(* IEC 61131-3 sources: Automation-Projects-Portfolio/Project1-TankLevelControl, 7 files *)

(* ---- DUT_Alarms.st ---- *)
TYPE DUT_Alarms :
STRUCT
		// Alarms setpoint
	rSetPointAlarm_HH : REAL := 90.0;
	rSetPointAlarm_H : REAL := 80.0;
	rSetPointAlarm_L : REAL := 20.0;
	rSetPointAlarm_LL : REAL := 10.0;

	//Alarm Status
	xAlarm_HH : BOOL;
	xAlarm_H : BOOL;
	xAlarm_L : BOOL ;
	xAlarm_LL : BOOL;

	//Sensor Fault
	xSensorFault : BOOL;
END_STRUCT
END_TYPE

(* ---- GVLInputs.st ---- *)
VAR_GLOBAL
	rLevelRaw : REAL; //Measured level from level transmitter
	xInletPumpRunFB : BOOL; //Feedback if inlet pump works
	xOutletPumpRunFB : BOOL; //Feedback if outlet pump works
	xEmergencyStop : BOOL := TRUE; //Emergency Button
END_VAR

(* ---- GVLOutputs.st ---- *)
VAR_GLOBAL
	xInletPumpStart : BOOL; //It is inlet pump start signal, if its contactor gets 24V DC from PLC, it will run
	xOutletPumpStart : BOOL; //It is outlet pump start signal, if its contactor gets 24V DC from PLC, it will run
	rValvePosition : REAL; //It is valve position which is decided by PID or an operator
END_VAR

(* ---- FB_ControlValve.st ---- *)
FUNCTION_BLOCK FB_ControlValve
VAR_INPUT
	xAutoMode : BOOL; // Auto = true, manual = false
	rAutoValvePosition : REAL; //Auto Valve position by PID
	rManualValvePosition : REAL; // Manual Valve Position by PID
	xSafetyClose : BOOL; //IF it is true, force valve to stop
END_VAR
VAR_OUTPUT
	rValvePosition : REAL; //ValvePosition is sent to control Valve
END_VAR
VAR
END_VAR

IF xSafetyClose THEN
	rValvePosition := 0.0; // Closed Valve
ELSIF xAutoMode THEN
	rValvePosition := rAutoValvePosition;
ELSE
	rValvePosition := rManualValvePosition;
END_IF

//Limit Valve Position
IF rValvePosition > 100.0 THEN
	rValvePosition := 100.0;
ELSIF rValvePosition < 0.0 THEN
	rValvePosition := 0.0;
END_IF

(* ---- FB_LevelControl.st ---- *)
FUNCTION_BLOCK FB_LevelControl
VAR_INPUT
	xAutoMode : BOOL; // TRUE = Auto FALSE = MANUAL
	rLevel : REAL; //Input from GVLInputs
	rSetPoint : REAL; //Target Level
	rKp : REAL := 2.0; // Proportianl gain in seconds;
	rTn : REAL := 10.0; //Integral time in seconds;
	rTv : REAL := 0.0;// DerivativeTime in seconds
	xResetAlarms : BOOL; //Reset after error is removed
END_VAR
VAR_OUTPUT
	rPidOutput : REAL;
	stAlarms : DUT_Alarms;
END_VAR
VAR
	PID : UTIL.PID;
	fbResetTrigger : R_TRIG; //Function block for reset
	xResetPulse : BOOL;
END_VAR

// 1. Reset for one cycle
fbResetTrigger ( CLK := xResetAlarms, Q => xResetPulse);

// 2. Sensor Fault Detection & Latched Reset
IF (rLevel < -2.0) OR (rLevel > 102.0) THEN
    stAlarms.xSensorFault := TRUE; // Latch Sensor Fault
ELSIF xResetPulse AND (rLevel >= 0.0) AND (rLevel <= 100.0) THEN
    stAlarms.xSensorFault := FALSE; // Reset Fault ONLY on 1-scan pulse AND safe level
END_IF

// 3. Latched High-High Alarm
IF (rLevel >= stAlarms.rSetPointAlarm_HH)  THEN
    stAlarms.xAlarm_HH := TRUE;
ELSIF xResetPulse AND (rLevel < stAlarms.rSetPointAlarm_HH) THEN
    stAlarms.xAlarm_HH := FALSE;
END_IF

// 4. Latched Low-Low Alarm
IF (rLevel <= stAlarms.rSetPointAlarm_LL) THEN
    stAlarms.xAlarm_LL := TRUE;
ELSIF xResetPulse AND (rLevel > stAlarms.rSetPointAlarm_LL) THEN
    stAlarms.xAlarm_LL := FALSE;
END_IF

// 5. Non-Latched Warning Alarms
stAlarms.xAlarm_H := (rLevel >= stAlarms.rSetPointAlarm_H);
stAlarms.xAlarm_L := (rLevel <= stAlarms.rSetPointAlarm_L);
//PID tuning parameters
PID(
	Actual := rLevel,
	SET_POINT := rSetPoint,
	Reset := xResetPulse,
	KP := rKp,
	TN := rTn,
	TV := rTv,
	Y_MIN := 0.0,
	Y_MAX := 100.0,
	Y => rPidOutput
);

//Checking Auto Mode
IF NOT xAutoMode OR stAlarms.xSensorFault THEN
	rPidOutput := 0.0;
END_IF

(* ---- FB_Pump.st ---- *)
FUNCTION_BLOCK FB_Pump
VAR_INPUT
	xAutoMode : BOOL; // Auto = TRUE, Manual = False;
	xAutoStartCmd : BOOL; //Start signal of auto mode
	xManStartCmd : BOOL; //Start signal of manual mode
	xInterlock : BOOL; //If it is true system is okay, there is no fault
	xFeedback : BOOL; //Feedback signal from motor
	tFeedbackDelay : TIME; //Allowed time to response
	xReset : BOOL; //If feedback error is handled so press reset button on hmi
END_VAR
VAR_OUTPUT
	xStartCmd : BOOL; //Start signal is sent to Motor
	xRunning : BOOL; // Confirmation of feedback
	xFeedbackError : BOOL; //if in spesific time if there is no feedback signal so there is error

END_VAR
VAR
	tFeedbackCountDown : TON; //Countdown for feedback signal
	fbResetTrigger : R_TRIG; //Function Block for Reset
	xResetPulse : BOOL; // Reset for one cycle
END_VAR

// 1. Reset Faults
fbResetTrigger(CLK := xReset, Q=> xResetPulse);
IF xResetPulse THEN
    xFeedbackError := FALSE;
END_IF

// 2. Safety & Mode Selection
IF xFeedbackError OR NOT xInterlock THEN
    xStartCmd := FALSE; // Block start command if there is a fault
ELSIF xAutoMode THEN
    xStartCmd := xAutoStartCmd;
ELSE
    xStartCmd := xManStartCmd;
END_IF

// 3. Feedback Checking
tFeedbackCountDown(IN := (xStartCmd AND NOT xFeedback), PT := tFeedbackDelay);

IF tFeedbackCountDown.Q THEN
    xFeedbackError := TRUE;
END_IF

// 4. Status Confirmation
xRunning := xFeedback;

(* ---- PLC_PRG.st ---- *)
PROGRAM PLC_PRG
VAR
	// Function Block Instnces
	fbLevelControl : FB_LevelControl;
	fbInletPump : FB_Pump;
	fbOutletPump : FB_Pump;
	fbControlValve : FB_ControlValve;

	//Permissive And SafetyClose
	xInletPermissive : BOOL;
	xOutletPermissive : BOOL;
	xValveSafetyClose : BOOL;

	//Manual mode commands
	xManualInletPumpStartCmd : BOOL;
	xManualOutletPumpStartCmd : BOOL;
	xManualValvePosition : REAL;
	//Inputs
	rSetPointHmi : REAL;
	xResetHMI : BOOL;

	//System Mode
	xSystemMode : BOOL := TRUE;
	xAlarm_HH: BOOL;
	xSensorFault: BOOL;
	xAlarm_LL: BOOL;
END_VAR

fbLevelControl(
	xAutoMode := xSystemMode,
	rLevel := GVLInputs.rLevelRaw,
	rSetPoint := rSetPointHmi,
	xResetAlarms := xResetHMI
);

xAlarm_HH := fbLevelControl.stAlarms.xAlarm_HH;
xAlarm_LL := fbLevelControl.stAlarms.xAlarm_LL;
xSensorFault := fbLevelControl.stAlarms.xSensorFault;

ACT_Interlock();

fbInletPump(
	xAutoMode := xSystemMode,
	xAutoStartCmd := (fbLevelControl.rPidOutput > 5.0),
	xManStartCmd := xManualInletPumpStartCmd,
	xInterlock := xInletPermissive,
	xFeedback := GVLInputs.xInletPumpRunFB,
	xReset := xResetHMI,
	xStartCmd => GVLOutputs.xInletPumpStart
);

fbOutletPump(
	xAutoMode := xSystemMode,
	xAutoStartCmd := TRUE,
	xManStartCmd := xManualOutletPumpStartCmd ,
	xInterlock := xOutletPermissive,
	xFeedback := GVLInputs.xOutletPumpRunFB,
	xReset := xResetHMI,
	xStartCmd => GVLOutputs.xOutletPumpStart
);
fbControlValve(
	xAutoMode := xSystemMode,
	rAutoValvePosition := fbLevelControl.rPidOutput,
	rManualValvePosition := xManualValvePosition,
	xSafetyClose := xValveSafetyClose,
	rValvePosition => GVLOutputs.rValvePosition
);
